FUNCTION_BLOCK TrajectoryGenerator
VAR_INPUT
END_VAR
VAR_OUTPUT
END_VAR
VAR
END_VAR

METHOD getTrajectory : ARRAY [0..100] OF RobotPoseSimple;
VAR_INPUT
	xWaypointList : ARRAY [0..100] OF RobotPoseSimple;
END_VAR

VAR
	trajectory : ARRAY [0..1000] OF RobotPoseSimple;
END_VAR
// calculate trajectory

getTrajectory := trajectory;
END_METHOD

END_FUNCTION_BLOCK

(* stored: Version 1.1.0.1, ProductVersion 3.1.4024.11
   POU TrajectoryGenerator: Id {8c501445-3a78-4866-be3e-a866b6d9ea9b}, SpecialFunc None
   Method getTrajectory: Id {a6aa5e76-ad3e-4cc3-b94a-7f5de5975f02} *)
